DATA_BLOCK "DB_G16OperationalCommand"
{ S7_Optimized_Access := 'TRUE' }
VERSION : 0.1
NON_RETAIN
   VAR
      Data : "UDT_G16OperationalCommand";
   END_VAR

BEGIN
END_DATA_BLOCK
